TYPE ST_Gear : //
STRUCT
	bEnable		                        :BOOL;	
	bGearOutMode                 :BOOL;
 
	bReady                            :BOOL;  
	bInGear		 	                   :BOOL;	
	bError				               :BOOL;			
END_STRUCT
END_TYPE

(* stored: Version 1.1.0.1, ProductVersion 3.1.4024.9
   DUT ST_Gear: Id {aa810c19-69e1-47db-a3dd-a67f9584c798} *)
